// TIA Portal project "FactoryIO_Template_S7-1200_V16_V16" (V16)
// Vorlageprojekt für das Buch mit Zielsystem S7-1200

(* hardware
DEVICE "S7-1200-Station_1"  S7-1200 Station
   slot 0: "Baugruppenträger_0"  Rack  V1.0
   slot 1: "PLC_1"  CPU 1211C DC/DC/DC  6ES7 211-1AE40-0XB0  V4.1
*)

// ===== PLC "PLC_1"  CPU 1211C DC/DC/DC =====

VAR_GLOBAL   // PLC tag table "Standard-Variablentabelle"
   "belt" AT %A0.0 : Bool;
   "start" AT %E0.0 : Bool;
   "stop" AT %E0.1 : Bool;
   "small" AT %I0.2 : Bool;
   "large" AT %I0.3 : Bool;
   "bl" AT %I0.4 : Bool;
   "fl" AT %I0.5 : Bool;
   "pusher" AT %Q0.1 : Bool;
   "x" AT %M0.0 : Bool;
   "y" AT %M0.1 : Bool;
   "Tag_2" AT %M0.2 : Bool;
   "z" AT %M0.5 : Bool;
   "s" AT %M3.0 : Bool;
   "Tag_1" AT %M3.1 : Bool;
END_VAR

FUNCTION "MHJ-PLC-Lab-Function-S71200" : Void   // FC9000, SCL
{ S7_Optimized_Access := 'TRUE' }
VERSION : 0.1
   VAR_TEMP
      rdTimeReturn : Int;
      outputTime : DTL;
      SyncVal : Byte;
      forVal : Int;
      forVal_2 : Int;
      Value : Byte;
   END_VAR
   VAR CONSTANT
      CompVal : Byte := 16#34;
      Value_01 : Byte := 16#11;
      Value_01_DW : DWord := 16#A165_D992;
      Value_02_DW : DWord := 16#58BE_4401;
   END_VAR
BEGIN

   #Value:=PEEK(area := 16#82,
        dbNumber := 0,
        byteOffset := 511);
   #Value := #Value + 1;

   POKE(area := 16#82,
        dbNumber := 0,
        byteOffset := 511,
        value := #Value);

   POKE(area:=16#81,
        dbNumber:=0,
        byteOffset:=1016,
        value:=#Value_01_DW);
   POKE(area := 16#81,
        dbNumber := 0,
        byteOffset := 1020,
        value := #Value_02_DW);

   POKE(area := 16#81,
        dbNumber := 0,
        byteOffset := 511,
        value := B#16#00);

   FOR #forVal := 0 TO 120 DO
       FOR #forVal_2:=0 TO 10 DO
           #rdTimeReturn:=RD_SYS_T(#outputTime);
           #rdTimeReturn := WR_SYS_T(#outputTime);
           #rdTimeReturn := RD_SYS_T(#outputTime);
           #rdTimeReturn := WR_SYS_T(#outputTime);
       END_FOR;
       #SyncVal:= PEEK(area := 16#81,
                      dbNumber := 0,
                      byteOffset := 511);
       IF #SyncVal = #CompVal THEN
          GOTO M_1;
       END_IF;
   END_FOR;
   RETURN;

   M_1:
   POKE(area := 16#81,
        dbNumber := 0,
        byteOffset := 511,
        value := B#16#0);
END_FUNCTION

ORGANIZATION_BLOCK "Main"   // OB1, LAD, ProgramCycle
TITLE = "Main Program Sweep (Cycle)"
{ S7_Optimized_Access := 'TRUE' }
VERSION : 0.1
   VAR_INPUT
      Initial_Call : Bool;   // Initial call of this OB
      Remanence : Bool;   // =True, if remanent data are available
   END_VAR
   VAR_TEMP   // added for the SCL form of the ladder/FBD networks
      _w1 : Bool;
   END_VAR
BEGIN

REGION Network 1: Konnektierungsbaustein für PLC-Lab
   // Im Netzwerk 1 wird der Konnektierungsbaustein für PLC-Lab aufgerufen.
   // Dieser Aufruf darf nicht entfernt werden!
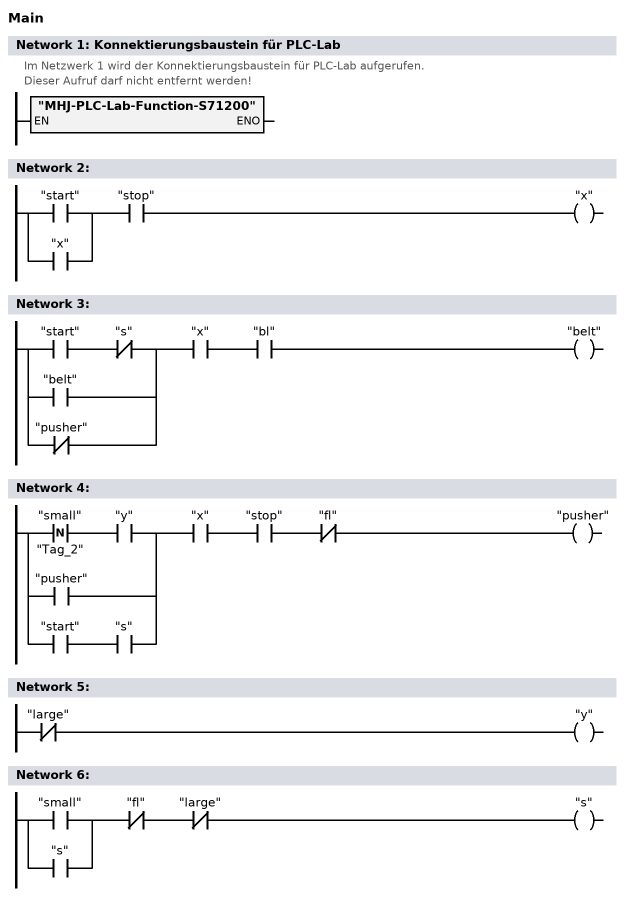
   RUNG wire#powerrail
      "MHJ-PLC-Lab-Function-S71200"()
   END_RUNG
   // the same network as SCL:
   "MHJ-PLC-Lab-Function-S71200"();
END_REGION

REGION Network 2
   RUNG wire#powerrail
      Contact( "start" )
      wire#w1
      Contact( "stop" )
      Coil( "x" )
   END_RUNG
   RUNG wire#powerrail
      Contact( "x" )
   END_RUNG wire#w1
   // the same network as SCL:
   "x" := ("start" OR "x") AND "stop";
END_REGION

REGION Network 3
   RUNG wire#powerrail
      Contact( "start" )
      I_Contact( "s" )
      wire#w1
      Contact( "x" )
      Contact( "bl" )
      Coil( "belt" )
   END_RUNG
   RUNG wire#powerrail
      Contact( "belt" )
   END_RUNG wire#w1
   RUNG wire#powerrail
      I_Contact( "pusher" )
   END_RUNG wire#w1
   // the same network as SCL:
   "belt" := (("start" AND NOT "s") OR "belt" OR NOT "pusher") AND "x" AND "bl";
END_REGION

REGION Network 4
   RUNG wire#powerrail
      N_Contact(operand := "small", bit := "Tag_2")
      Contact( "y" )
      wire#w1
      Contact( "x" )
      Contact( "stop" )
      I_Contact( "fl" )
      Coil( "pusher" )
   END_RUNG
   RUNG wire#powerrail
      Contact( "pusher" )
   END_RUNG wire#w1
   RUNG wire#powerrail
      Contact( "start" )
      Contact( "s" )
   END_RUNG wire#w1
   // the same network as SCL:
   #_w1 := NOT "small" AND "Tag_2";   // falling edge of "small"
   "Tag_2" := "small";
   "pusher" := ((#_w1 AND "y") OR "pusher" OR ("start" AND "s")) AND "x" AND "stop" AND NOT "fl";
END_REGION

REGION Network 5
   RUNG wire#powerrail
      I_Contact( "large" )
      Coil( "y" )
   END_RUNG
   // the same network as SCL:
   "y" := NOT "large";
END_REGION

REGION Network 6
   RUNG wire#powerrail
      Contact( "small" )
      wire#w1
      I_Contact( "fl" )
      I_Contact( "large" )
      Coil( "s" )
   END_RUNG
   RUNG wire#powerrail
      Contact( "s" )
   END_RUNG wire#w1
   // the same network as SCL:
   "s" := ("small" OR "s") AND NOT "fl" AND NOT "large";
END_REGION
END_ORGANIZATION_BLOCK